FUNCTION_BLOCK CM_Merge2E2USINT (* Basic Function Block Type *)
  (* Standard: 61499-2 *)
  (* Version 0.0, 2014-09-04, EQUEROL, UJI *)
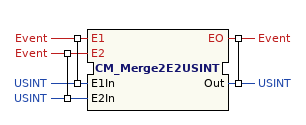
  EVENT_INPUT
    E1 WITH E1In; (* Event 1 to merge *)
    E2 WITH E2In; (* Event 2 to merge *)
  END_EVENT
  EVENT_OUTPUT
    EO WITH Out; (* Event Output *)
  END_EVENT
  VAR_INPUT
    E1In : USINT;
    E2In : USINT;
  END_VAR
  VAR_OUTPUT
    Out : USINT; (* Merge output *)
  END_VAR
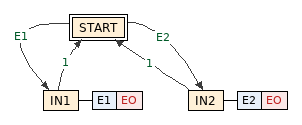
  EC_STATES
    START; (* Initial State *)
    IN1 : E1 -> EO;
    IN2 : E2 -> EO;
  END_STATES
  EC_TRANSITIONS
    START TO IN1 := E1;
    START TO IN2 := E2;
    IN1 TO START := 1;
    IN2 TO START := 1;
  END_TRANSITIONS
  ALGORITHM E1 IN ST: (* new algorithm *)
Out := E1In;
  END_ALGORITHM
  ALGORITHM E2 IN ST: (* new algorithm *)
Out := E2In;
  END_ALGORITHM
END_FUNCTION_BLOCK
